// TIA Portal V17 export
// export: Created 2025-05-06T14:29:00.5141896Z, ExportSetting WithDefaults, DisplayName Totally Integrated Automation Portal, DisplayVersion V17 Update 8, DisplayName TIA Portal Openness, DisplayVersion V17 Update 8, DisplayName TIA Portal Version Control Interface, DisplayVersion V17, DisplayName SINAMICS Startdrive Advanced, DisplayVersion V17 SP2, DisplayName SINAMICS Startdrive G110M, G120, G120C, G120D, G120P, G115D, DisplayVersion V17 SP2, DisplayName SINAMICS Startdrive G130, G150, S120, S150, SINAMICS MV, S210, DisplayVersion V17 SP2, DisplayName STEP 7 Professional, DisplayVersion V17 Update 8, DisplayName SINUMERIK ONE STEP 7 Toolbox, DisplayVersion V17 Update 12, DisplayName SINUMERIK 840D sl STEP 7 Toolbox, DisplayVersion V17 Update 12, DisplayName STEP 7 Safety, DisplayVersion V17 Update 6, DisplayName WinCC Advanced, DisplayVersion V17 Update 8
DATA_BLOCK "DB7241_PROCESS_PARAMETERS"   // DB7241
{ S7_Optimized_Access := 'FALSE'; DB_Accessible_From_OPC_UA := 'FALSE' }
VERSION : 0.1
// stored: AutoNumber false, DBAccessibleFromOPCUA false, DBAccessibleFromWebserver true, IsOnlyStoredInLoadMemory false, IsWriteProtectedInAS false
   VAR RETAIN
      UNIT_1 : Struct
         POSITIONS : Struct
            START_POS_RS_FACE : Real := 177.0;   // UNIT 1 START POSITION RS FACE
            START_POS_NS_FACE : Real;   // UNIT 1 START POSITION NS FACE
            FINAL_POSITION : Real;   // UNIT 1 FINAL POSITION POSITION
            WORKING_DISTANCE : Real;   // UNIT 1 WORKING DISTANCE POSITION
            RADIAL_ANGLE : Real;   // UNIT 1 RADIAL ANGLE POSITION
            TANGENTIAL_ANGLE : Real;   // UNIT 1 TANGENTIAL ANGLE POSITION
            CAMERA_CALIBATION : Real;   // UNIT 1 CAMERA CALIBRATION POSITION
            CAMERA_CALIB_MOV : Real;   // UNIT 1 CAMERA CALIBRATION MOVEMENT
         END_STRUCT;
         FEEDRATES : Struct
            TANGENT_FEED : Int;   // UNIT 1 TANGENT FEED
            RADIAL_FEED : Real;   // UNIT 1 RADIAL FEED
         END_STRUCT;
         LASER : Struct
            PROCESSING : Int;   // UNIT 1 LASER PROCESSING TYPE
            POWER_PORTION_CORE : Int;   // UNIT 1 LASER POWER PORTION CORE
            POWER_DISTRIBUTION : Int;   // UNIT 1 LASER POWER DISTRIBUTION
            POWER : Int;   // UNIT 1 LASER POWER
            PROTECTION_GAS : Int;   // UNIT 1 LASER PROTECTION GAS
         END_STRUCT;
         POWDER_FEEDERS : Struct
            FEEDER_1 : Struct
               CARRIER_GAS_LINE_1 : Int;   // UNIT 1 POWDER FEEDER 1 LINE 1 CARRIER GAS
               CARRIER_GAS_LINE_2 : Int;   // UNIT 1 POWDER FEEDER 1 LINE 2 CARRIER GAS
               DISK_SPEED_LINE_1 : Int;   // UNIT 1 POWDER FEEDER 1 LINE 1 DISK SPEED
               DISK_SPEED_LINE_2 : Int;   // UNIT 1 POWDER FEEDER 1 LINE 2 DISK SPEED
               STIRRER_SPEED_LINE_1 : Int;   // UNIT 1 POWDER FEEDER 1 LINE 1 STIRRER SPEED
               STIRRER_SPEED_LINE_2 : Int;   // UNIT 1 POWDER FEEDER 1 LINE 2 STIRRER SPEED
            END_STRUCT;
         END_STRUCT;
         LIMITS : Struct
            START_POS_RS_FACE_LOW_LIM : Real := 177.0;   // UNIT 1 START POSITION RS FACE LOW LIMIT
            START_POS_RS_FACE_UP_LIM : Real := 197.0;   // UNIT 1 START POSITION RS FACE UPPER LIMIT
            START_POS_NS_FACE_LOW_LIM : Real := 177.0;   // UNIT 1 START POSITION NS FACE LOW LIMIT
            START_POS_NS_FACE_UP_LIM : Real := 197.0;   // UNIT 1 START POSITION NS FACE UPPER LIMIT
            FINAL_POS_LOW_LIM : Real := 286.0;   // UNIT 1 FINAL POSITION LOW LIMIT
            FINAL_POS_UP_LIM : Real := 306.0;   // UNIT 1 FINAL POSITION UPPER LIMIT
            TANGENT_FEED_LOW_LIM : Int := 100;   // UNIT 1 TANGENT FEED LOW LIMIT
            TANGENT_FEED_UP_LIM : Int := 150;   // UNIT 1 TANGENT FEED UPPER LIMIT
            RADIAL_FEED_LOW_LIM : Real := 0.0;   // UNIT 1 RADIAL FEED LOW LIMIT
            RADIAL_FEED_UP_LIM : Real := 1.0;   // UNIT 1 RADIAL FEED UPPER LIMIT
            POWER_PORTION_CORE_LOW_LIM : Int := 0;   // UNIT 1 POWER PORTION CORE LOW LIMIT
            POWER_PORTION_CORE_UP_LIM : Int := 100;   // UNIT 1 POWER PORTION CORE UPPER LIMIT
            POWER_DISTRIBUTION_LOW_LIM : Int := 0;   // UNIT 1 POWER DISTRIBUTION LOW LIMIT
            POWER_DISTRIBUTION_UP_LIM : Int := 50;   // UNIT 1 POWER DISTRIBUTION UPPER LIMIT
            POWER_LOW_LIM : Int := 0;   // UNIT 1 POWER LOW LIMIT
            POWER_UP_LIM : Int := 20000;   // UNIT 1 POWER UPPER LIMIT
            WORKING_DISTANCE_LOW_LIM : Real := 26.0;   // UNIT 1 WORKING DISTANCE LOW LIMIT
            WORKING_DISTANCE_UP_LIM : Real := 32.0;   // UNIT 1 WORKING DISTANCE UPPER LIMIT
            RADIAL_ANGLE_LOW_LIM : Real := 0.0;   // UNIT 1 RADIAL ANGLE LOW LIMIT
            RADIAL_ANGLE_UP_LIM : Real := 10.0;   // UNIT 1 RADIAL ANGLE UPPER LIMIT
            TANGENCIAL_ANGLE_LOW_LIM : Real := 0.0;   // UNIT 1 TANGENCIAL ANGLE LOW LIMIT
            TANGENCIAL_ANGLE_UP_LIM : Real := 15.0;   // UNIT 1 TANGENCIAL ANGLE UPPER LIMIT
            CAMERA_CALIB_POS_LOW_LIM : Real := 177.0;   // UNIT 1 CAMERA CALIBRATION POSITION LOW LIMIT
            CAMERA_CALIB_POS_UP_LIM : Real := 306.0;   // UNIT 1 CAMERA CALIBRATION POSITION UPPER LIMIT
            CAMERA_CALIB_MOV_LOW_LIM : Real := 0.0;   // UNIT 1 CAMERA CALIBRATION MOVEMENT LOW LIMIT
            CAMERA_CALIB_MOV_UP_LIM : Real := 6.0;   // UNIT 1 CAMERA CALIBRATION MOVEMENT UPPER LIMIT
            PF_1_CARRIER_GAS_LINE_1_LOW_LIM : Int := 0;   // UNIT 1 POWDER FEEDER 1 LINE 1 CARRIER GAS LOWER LIMIT
            PF_1_CARRIER_GAS_LINE_1_UP_LIM : Int := 30;   // UNIT 1 POWDER FEEDER 1 LINE 1 CARRIER GAS UPPER LIMIT
            PF_1_CARRIER_GAS_LINE_2_LOW_LIM : Int := 0;   // UNIT 1 POWDER FEEDER 1 LINE 2 CARRIER GAS LOWER LIMIT
            PF_1_CARRIER_GAS_LINE_2_UP_LIM : Int := 30;   // UNIT 1 POWDER FEEDER 1 LINE 2 CARRIER GAS UPPER LIMIT
            PF_1_DISK_SPEED_LINE_1_LOW_LIM : Int := 0;   // UNIT 1 POWDER FEEDER 1 LINE 1 DISK SPEED LOWER LIMIT
            PF_1_DISK_SPEED_LINE_1_UP_LIM : Int := 100;   // UNIT 1 POWDER FEEDER 1 LINE 1 DISK SPEED UPPER LIMIT
            PF_1_DISK_SPEED_LINE_2_LOW_LIM : Int := 0;   // UNIT 1 POWDER FEEDER 1 LINE 2 DISK SPEED LOWER LIMIT
            PF_1_DISK_SPEED_LINE_2_UP_LIM : Int := 100;   // UNIT 1 POWDER FEEDER 1 LINE 2 DISK SPEED UPPER LIMIT
            PF_1_STIRRER_SPEED_LINE_1_LOW_LIM : Int := 0;   // UNIT 1 POWDER FEEDER 1 LINE 1 STIRRER SPEED LOWER LIMIT
            PF_1_STIRRER_SPEED_LINE_1_UP_LIM : Int := 100;   // UNIT 1 POWDER FEEDER 1 LINE 1 STIRRER SPEED UPPER LIMIT
            PF_1_STIRRER_SPEED_LINE_2_LOW_LIM : Int := 0;   // UNIT 1 POWDER FEEDER 1 LINE 2 STIRRER SPEED LOWER LIMIT
            PF_1_STIRRER_SPEED_LINE_2_UP_LIM : Int := 100;   // UNIT 1 POWDER FEEDER 1 LINE 2 STIRRER SPEED UPPER LIMIT
            PROTECTION_GAS_LOW_LIM : Int := 0;   // UNIT 1 PROTECTION GAS LOWER LIMIT
            PROTECTION_GAS_UP_LIM : Int := 50;   // UNIT 1 PROTECTION UPPER LIMIT
         END_STRUCT;
      END_STRUCT;
      UNIT_2 : Struct
         POSITIONS : Struct
            START_POS_RS_FACE : Real := 178.0;   // UNIT 2 START POSITION RS FACE
            START_POS_NS_FACE : Real;   // UNIT 2 START POSITION NS FACE
            FINAL_POSITION : Real;   // UNIT 2 FINAL POSITION POSITION
            WORKING_DISTANCE : Real;   // UNIT 2 WORKING DISTANCE POSITION
            RADIAL_ANGLE : Real;   // UNIT 2 RADIAL ANGLE POSITION
            TANGENTIAL_ANGLE : Real;   // UNIT 2 TANGENTIAL ANGLE POSITION
            CAMERA_CALIBATION : Real;   // UNIT 2 CAMERA CALIBRATION POSITION
            CAMERA_CALIB_MOV : Real;   // UNIT 2 CAMERA CALIBRATION MOVEMENT
         END_STRUCT;
         FEEDRATES : Struct
            TANGENT_FEED : Int;   // UNIT 2 TANGENT FEED
            RADIAL_FEED : Real;   // UNIT 2 RADIAL FEED
         END_STRUCT;
         LASER : Struct
            PROCESSING : Int;   // UNIT 2 LASER PROCESSING TYPE
            POWER_PORTION_CORE : Int;   // UNIT 2 LASER POWER PORTION CORE
            POWER_DISTRIBUTION : Int;   // UNIT 2 LASER POWER DISTRIBUTION
            POWER : Int;   // UNIT 2 LASER POWER
            PROTECTION_GAS : Int;   // UNIT 2 LASER PROTECTION GAS
         END_STRUCT;
         POWDER_FEEDERS : Struct
            FEEDER_1 : Struct
               CARRIER_GAS_LINE_1 : Int;   // UNIT 2 POWDER FEEDER 1 LINE 1 CARRIER GAS
               CARRIER_GAS_LINE_2 : Int;   // UNIT 2 POWDER FEEDER 1 LINE 2 CARRIER GAS
               DISK_SPEED_LINE_1 : Int;   // UNIT 2 POWDER FEEDER 1 LINE 1 DISK SPEED
               DISK_SPEED_LINE_2 : Int;   // UNIT 2 POWDER FEEDER 1 LINE 2 DISK SPEED
               STIRRER_SPEED_LINE_1 : Int;   // UNIT 2 POWDER FEEDER 1 LINE 1 STIRRER SPEED
               STIRRER_SPEED_LINE_2 : Int;   // UNIT 2 POWDER FEEDER 1 LINE 2 STIRRER SPEED
            END_STRUCT;
            FEEDER_2 : Struct
               CARRIER_GAS_LINE_1 : Int;   // UNIT 2 POWDER FEEDER 2 LINE 1 CARRIER GAS
               CARRIER_GAS_LINE_2 : Int;   // UNIT 2 POWDER FEEDER 2 LINE 2 CARRIER GAS
               DISK_SPEED_LINE_1 : Int;   // UNIT 2 POWDER FEEDER 2 LINE 1 DISK SPEED
               DISK_SPEED_LINE_2 : Int;   // UNIT 2 POWDER FEEDER 2 LINE 2 DISK SPEED
               STIRRER_SPEED_LINE_1 : Int;   // UNIT 2 POWDER FEEDER 2 LINE 1 STIRRER SPEED
               STIRRER_SPEED_LINE_2 : Int;   // UNIT 2 POWDER FEEDER 2 LINE 2 STIRRER SPEED
            END_STRUCT;
         END_STRUCT;
         LIMITS : Struct
            START_POS_RS_FACE_LOW_LIM : Real := 177.0;   // UNIT 2 START POSITION RS FACE LOW LIMIT
            START_POS_RS_FACE_UP_LIM : Real := 197.0;   // UNIT 2 START POSITION RS FACE UPPER LIMIT
            START_POS_NS_FACE_LOW_LIM : Real := 177.0;   // UNIT 2 START POSITION NS FACE LOW LIMIT
            START_POS_NS_FACE_UP_LIM : Real := 197.0;   // UNIT 2 START POSITION NS FACE UPPER LIMIT
            FINAL_POS_LOW_LIM : Real := 286.0;   // UNIT 2 FINAL POSITION LOW LIMIT
            FINAL_POS_UP_LIM : Real := 306.0;   // UNIT 2 FINAL POSITION UPPER LIMIT
            TANGENT_FEED_LOW_LIM : Int := 100;   // UNIT 2 TANGENT FEED LOW LIMIT
            TANGENT_FEED_UP_LIM : Int := 150;   // UNIT 2 TANGENT FEED UPPER LIMIT
            RADIAL_FEED_LOW_LIM : Real := 0.0;   // UNIT 2 RADIAL FEED LOW LIMIT
            RADIAL_FEED_UP_LIM : Real := 1.0;   // UNIT 2 RADIAL FEED UPPER LIMIT
            POWER_PORTION_CORE_LOW_LIM : Int := 0;   // UNIT 2 POWER PORTION CORE LOW LIMIT
            POWER_PORTION_CORE_UP_LIM : Int := 100;   // UNIT 2 POWER PORTION CORE UPPER LIMIT
            POWER_DISTRIBUTION_LOW_LIM : Int := 0;   // UNIT 2 POWER DISTRIBUTION LOW LIMIT
            POWER_DISTRIBUTION_UP_LIM : Int := 50;   // UNIT 2 POWER DISTRIBUTION UPPER LIMIT
            POWER_LOW_LIM : Int := 0;   // UNIT 2 POWER LOW LIMIT
            POWER_UP_LIM : Int := 20000;   // UNIT 2 POWER UPPER LIMIT
            WORKING_DISTANCE_LOW_LIM : Real := 26.0;   // UNIT 2 WORKING DISTANCE LOW LIMIT
            WORKING_DISTANCE_UP_LIM : Real := 32.0;   // UNIT 2 WORKING DISTANCE UPPER LIMIT
            RADIAL_ANGLE_LOW_LIM : Real := 0.0;   // UNIT 2 RADIAL ANGLE LOW LIMIT
            RADIAL_ANGLE_UP_LIM : Real := 10.0;   // UNIT 2 RADIAL ANGLE UPPER LIMIT
            TANGENCIAL_ANGLE_LOW_LIM : Real := 0.0;   // UNIT 2 TANGENCIAL ANGLE LOW LIMIT
            TANGENCIAL_ANGLE_UP_LIM : Real := 15.0;   // UNIT 2 TANGENCIAL ANGLE UPPER LIMIT
            CAMERA_CALIB_POS_LOW_LIM : Real := 177.0;   // UNIT 2 CAMERA CALIBRATION POSITION LOW LIMIT
            CAMERA_CALIB_POS_UP_LIM : Real := 306.0;   // UNIT 2 CAMERA CALIBRATION POSITION UPPER LIMIT
            CAMERA_CALIB_MOV_LOW_LIM : Real := 0.0;   // UNIT 2 CAMERA CALIBRATION MOVEMENT LOW LIMIT
            CAMERA_CALIB_MOV_UP_LIM : Real := 6.0;   // UNIT 2 CAMERA CALIBRATION MOVEMENT UPPER LIMIT
            PF_1_CARRIER_GAS_LINE_1_LOW_LIM : Int := 0;   // UNIT 2 POWDER FEEDER 1 LINE 1 CARRIER GAS LOWER LIMIT
            PF_1_CARRIER_GAS_LINE_1_UP_LIM : Int := 30;   // UNIT 2 POWDER FEEDER 1 LINE 1 CARRIER GAS UPPER LIMIT
            PF_1_CARRIER_GAS_LINE_2_LOW_LIM : Int := 0;   // UNIT 2 POWDER FEEDER 1 LINE 2 CARRIER GAS LOWER LIMIT
            PF_1_CARRIER_GAS_LINE_2_UP_LIM : Int := 30;   // UNIT 2 POWDER FEEDER 1 LINE 2 CARRIER GAS UPPER LIMIT
            PF_1_DISK_SPEED_LINE_1_LOW_LIM : Int := 0;   // UNIT 2 POWDER FEEDER 1 LINE 1 DISK SPEED LOWER LIMIT
            PF_1_DISK_SPEED_LINE_1_UP_LIM : Int := 100;   // UNIT 2 POWDER FEEDER 1 LINE 1 DISK SPEED UPPER LIMIT
            PF_1_DISK_SPEED_LINE_2_LOW_LIM : Int := 0;   // UNIT 2 POWDER FEEDER 1 LINE 2 DISK SPEED LOWER LIMIT
            PF_1_DISK_SPEED_LINE_2_UP_LIM : Int := 100;   // UNIT 2 POWDER FEEDER 1 LINE 2 DISK SPEED UPPER LIMIT
            PF_1_STIRRER_SPEED_LINE_1_LOW_LIM : Int := 0;   // UNIT 2 POWDER FEEDER 1 LINE 1 STIRRER SPEED LOWER LIMIT
            PF_1_STIRRER_SPEED_LINE_1_UP_LIM : Int := 100;   // UNIT 2 POWDER FEEDER 1 LINE 1 STIRRER SPEED UPPER LIMIT
            PF_1_STIRRER_SPEED_LINE_2_LOW_LIM : Int := 0;   // UNIT 2 POWDER FEEDER 1 LINE 2 STIRRER SPEED LOWER LIMIT
            PF_1_STIRRER_SPEED_LINE_2_UP_LIM : Int := 100;   // UNIT 2 POWDER FEEDER 1 LINE 2 STIRRER SPEED UPPER LIMIT
            PF_2_CARRIER_GAS_LINE_1_LOW_LIM : Int := 0;   // UNIT 2 POWDER FEEDER 2 LINE 1 CARRIER GAS LOWER LIMIT
            PF_2_CARRIER_GAS_LINE_1_UP_LIM : Int := 30;   // UNIT 2 POWDER FEEDER 2 LINE 1 CARRIER GAS UPPER LIMIT
            PF_2_CARRIER_GAS_LINE_2_LOW_LIM : Int := 0;   // UNIT 2 POWDER FEEDER 2 LINE 2 CARRIER GAS LOWER LIMIT
            PF_2_CARRIER_GAS_LINE_2_UP_LIM : Int := 30;   // UNIT 2 POWDER FEEDER 2 LINE 2 CARRIER GAS UPPER LIMIT
            PF_2_DISK_SPEED_LINE_1_LOW_LIM : Int := 0;   // UNIT 2 POWDER FEEDER 2 LINE 1 DISK SPEED LOWER LIMIT
            PF_2_DISK_SPEED_LINE_1_UP_LIM : Int := 100;   // UNIT 2 POWDER FEEDER 2 LINE 1 DISK SPEED UPPER LIMIT
            PF_2_DISK_SPEED_LINE_2_LOW_LIM : Int := 0;   // UNIT 2 POWDER FEEDER 2 LINE 2 DISK SPEED LOWER LIMIT
            PF_2_DISK_SPEED_LINE_2_UP_LIM : Int := 100;   // UNIT 2 POWDER FEEDER 2 LINE 2 DISK SPEED UPPER LIMIT
            PF_2_STIRRER_SPEED_LINE_1_LOW_LIM : Int := 0;   // UNIT 2 POWDER FEEDER 2 LINE 1 STIRRER SPEED LOWER LIMIT
            PF_2_STIRRER_SPEED_LINE_1_UP_LIM : Int := 100;   // UNIT 2 POWDER FEEDER 2 LINE 1 STIRRER SPEED UPPER LIMIT
            PF_2_STIRRER_SPEED_LINE_2_LOW_LIM : Int := 0;   // UNIT 2 POWDER FEEDER 2 LINE 2 STIRRER SPEED LOWER LIMIT
            PF_2_STIRRER_SPEED_LINE_2_UP_LIM : Int := 100;   // UNIT 2 POWDER FEEDER 2 LINE 2 STIRRER SPEED UPPER LIMIT
            PROTECTION_GAS_LOW_LIM : Int := 0;   // UNIT 2 PROTECTION GAS LOWER LIMIT
            PROTECTION_GAS_UP_LIM : Int := 50;   // UNIT 2 PROTECTION UPPER LIMIT
         END_STRUCT;
      END_STRUCT;
   END_VAR
BEGIN
END_DATA_BLOCK
